{attribute 'pack_mode' := '1'}
TYPE TGiver :
	STRUCT
		bHasGiven		: BOOL;		(* Part has been given *)
		bPartDataReady	: BOOL;
		TPartData		: TPartData;
	END_STRUCT
END_TYPE

(* stored: Version 1.1.0.1, ProductVersion 3.1.4022.12
   DUT TGiver: Id {506892c3-ab28-4f9e-a361-1e9ad3d40c13} *)
